// TIA Portal V16 export
// export: Created 2022-11-17T15:49:28.7490525Z, ExportSetting WithDefaults, DisplayName Totally Integrated Automation Portal, DisplayVersion V16 Update 6, DisplayName TIA Portal Version Control Interface, DisplayVersion V16 Update 2, DisplayName TIA Portal Openness, DisplayVersion V16 Update 6, DisplayName SINAMICS Startdrive Advanced, DisplayVersion V16 Update 5, DisplayName SINAMICS Startdrive G130, G150, S120, S150, SINAMICS MV, S210, DisplayVersion V16 Update 5, DisplayName SINAMICS Startdrive G110M, G120, G120C, G120D, G120P, G115D, DisplayVersion V16 Update 5, DisplayName STEP 7 Professional, DisplayVersion V16 Update 6, DisplayName STEP 7 Safety, DisplayVersion V16, DisplayName WinCC Advanced, DisplayVersion V16 Update 6
FUNCTION "FC78_Conveyor_1_IN_1_OUT_REVERSE" : Void   // FC78, LAD
TITLE = Conveyor_1_IN_1_OUT
{ S7_Optimized_Access := 'TRUE' }
VERSION : 0.1
// stored: AutoNumber false, IsIECCheckEnabled false, SetENOAutomatically false, UDAEnableTagReadback false
   VAR_TEMP   // added for the SCL form of the ladder/FBD networks
      _w1 : Bool;
   END_VAR
BEGIN

REGION Network 1: Manual operation for conveyor
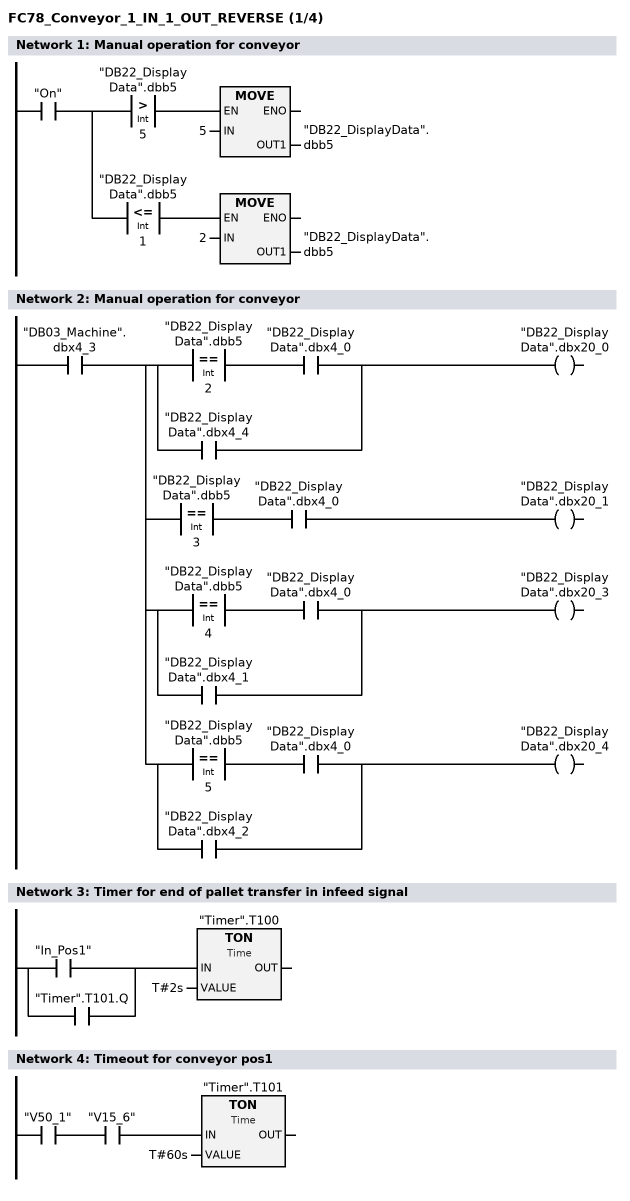
   RUNG wire#powerrail
      Contact( "On" )
      wire#w1
      { S7_Templates := "SrcType := Int" } GT_Contact(in1 := "DB22_DisplayData".dbb5, in2 := 5)
      { S7_GenerateENO := "TRUE" } Move(in := 5, out1 => "DB22_DisplayData".dbb5)
   END_RUNG
   RUNG wire#w1
      { S7_Templates := "SrcType := Int" } LE_Contact(in1 := "DB22_DisplayData".dbb5, in2 := 1)
      { S7_GenerateENO := "TRUE" } Move(in := 2, out1 => "DB22_DisplayData".dbb5)
   END_RUNG
   // the same network as SCL:
   IF "On" AND ("DB22_DisplayData".dbb5 > 5) THEN "DB22_DisplayData".dbb5 := 5; END_IF;
   IF "On" AND ("DB22_DisplayData".dbb5 <= 1) THEN "DB22_DisplayData".dbb5 := 2; END_IF;
END_REGION

REGION Network 2: Manual operation for conveyor
   RUNG wire#powerrail
      Contact( "DB03_Machine".dbx4_3 )
      wire#w1
      { S7_Templates := "SrcType := Int" } EQ_Contact(in1 := "DB22_DisplayData".dbb5, in2 := 2)
      Contact( "DB22_DisplayData".dbx4_0 )
      wire#w2
      Coil( "DB22_DisplayData".dbx20_0 )
   END_RUNG
   RUNG wire#w1
      Contact( "DB22_DisplayData".dbx4_4 )
   END_RUNG wire#w2
   RUNG wire#w1
      { S7_Templates := "SrcType := Int" } EQ_Contact(in1 := "DB22_DisplayData".dbb5, in2 := 3)
      Contact( "DB22_DisplayData".dbx4_0 )
      Coil( "DB22_DisplayData".dbx20_1 )
   END_RUNG
   RUNG wire#w1
      { S7_Templates := "SrcType := Int" } EQ_Contact(in1 := "DB22_DisplayData".dbb5, in2 := 4)
      Contact( "DB22_DisplayData".dbx4_0 )
      wire#w3
      Coil( "DB22_DisplayData".dbx20_3 )
   END_RUNG
   RUNG wire#w1
      Contact( "DB22_DisplayData".dbx4_1 )
   END_RUNG wire#w3
   RUNG wire#w1
      { S7_Templates := "SrcType := Int" } EQ_Contact(in1 := "DB22_DisplayData".dbb5, in2 := 5)
      Contact( "DB22_DisplayData".dbx4_0 )
      wire#w4
      Coil( "DB22_DisplayData".dbx20_4 )
   END_RUNG
   RUNG wire#w1
      Contact( "DB22_DisplayData".dbx4_2 )
   END_RUNG wire#w4
   // the same network as SCL:
   "DB22_DisplayData".dbx20_0 := "DB03_Machine".dbx4_3 AND ((("DB22_DisplayData".dbb5 = 2) AND "DB22_DisplayData".dbx4_0) OR "DB22_DisplayData".dbx4_4);
   "DB22_DisplayData".dbx20_1 := "DB03_Machine".dbx4_3 AND ("DB22_DisplayData".dbb5 = 3) AND "DB22_DisplayData".dbx4_0;
   "DB22_DisplayData".dbx20_3 := "DB03_Machine".dbx4_3 AND ((("DB22_DisplayData".dbb5 = 4) AND "DB22_DisplayData".dbx4_0) OR "DB22_DisplayData".dbx4_1);
   "DB22_DisplayData".dbx20_4 := "DB03_Machine".dbx4_3 AND ((("DB22_DisplayData".dbb5 = 5) AND "DB22_DisplayData".dbx4_0) OR "DB22_DisplayData".dbx4_2);
END_REGION

REGION Network 3: Timer for end of pallet transfer in infeed signal
   "Timer".T100.TON(IN := "In_Pos1" OR "Timer".T101.Q, PT := T#2s);   // TON coil
END_REGION

REGION Network 4: Timeout for conveyor pos1
   "Timer".T101.TON(IN := "V50_1" AND "V15_6", PT := T#60s);   // TON coil
END_REGION

REGION Network 5: Time to load with forklift
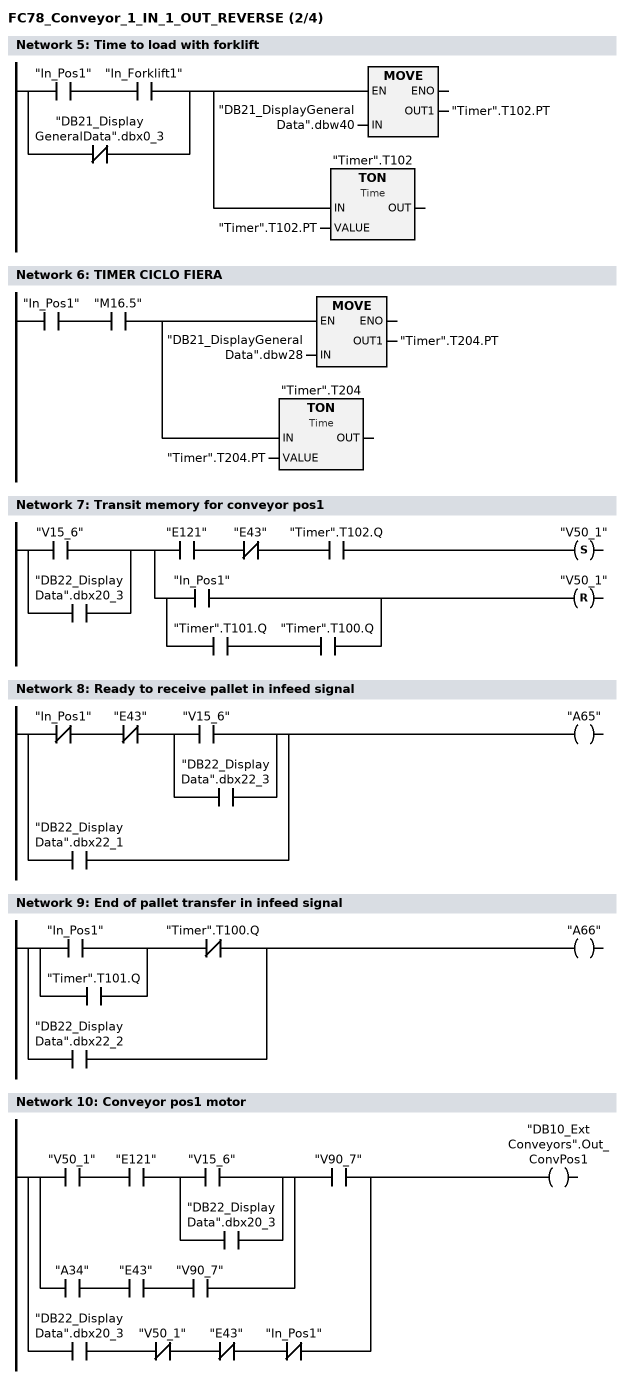
   #_w1 := ("In_Pos1" AND "In_Forklift1") OR NOT "DB21_DisplayGeneralData".dbx0_3;
   IF #_w1 THEN "Timer".T102.PT := "DB21_DisplayGeneralData".dbw40; END_IF;
   "Timer".T102.TON(IN := #_w1, PT := "Timer".T102.PT);   // TON coil
END_REGION

REGION Network 6: TIMER CICLO FIERA
   #_w1 := "In_Pos1" AND "M16.5";
   IF #_w1 THEN "Timer".T204.PT := "DB21_DisplayGeneralData".dbw28; END_IF;
   "Timer".T204.TON(IN := #_w1, PT := "Timer".T204.PT);   // TON coil
END_REGION

REGION Network 7: Transit memory for conveyor pos1
   RUNG wire#powerrail
      Contact( "V15_6" )
      wire#w1
      Contact( "E121" )
      I_Contact( "E43" )
      Contact( "Timer".T102.Q )
      S_Coil( "V50_1" )
   END_RUNG
   RUNG wire#powerrail
      Contact( "DB22_DisplayData".dbx20_3 )
   END_RUNG wire#w1
   RUNG wire#w1
      Contact( "In_Pos1" )
      wire#w2
      R_Coil( "V50_1" )
   END_RUNG
   RUNG wire#w1
      Contact( "Timer".T101.Q )
      Contact( "Timer".T100.Q )
   END_RUNG wire#w2
   // the same network as SCL:
   #_w1 := "V15_6" OR "DB22_DisplayData".dbx20_3;
   IF #_w1 AND "E121" AND NOT "E43" AND "Timer".T102.Q THEN "V50_1" := TRUE; END_IF;
   IF #_w1 AND ("In_Pos1" OR ("Timer".T101.Q AND "Timer".T100.Q)) THEN "V50_1" := FALSE; END_IF;
END_REGION

REGION Network 8: Ready to receive pallet in infeed signal
   RUNG wire#powerrail
      I_Contact( "In_Pos1" )
      I_Contact( "E43" )
      wire#w1
      Contact( "V15_6" )
      wire#w2
      Coil( "A65" )
   END_RUNG
   RUNG wire#w1
      Contact( "DB22_DisplayData".dbx22_3 )
   END_RUNG wire#w2
   RUNG wire#powerrail
      Contact( "DB22_DisplayData".dbx22_1 )
   END_RUNG wire#w2
   // the same network as SCL:
   "A65" := (NOT "In_Pos1" AND NOT "E43" AND ("V15_6" OR "DB22_DisplayData".dbx22_3)) OR "DB22_DisplayData".dbx22_1;
END_REGION

REGION Network 9: End of pallet transfer in infeed signal
   RUNG wire#powerrail
      Contact( "In_Pos1" )
      wire#w1
      I_Contact( "Timer".T100.Q )
      wire#w2
      Coil( "A66" )
   END_RUNG
   RUNG wire#powerrail
      Contact( "Timer".T101.Q )
   END_RUNG wire#w1
   RUNG wire#powerrail
      Contact( "DB22_DisplayData".dbx22_2 )
   END_RUNG wire#w2
   // the same network as SCL:
   "A66" := (("In_Pos1" OR "Timer".T101.Q) AND NOT "Timer".T100.Q) OR "DB22_DisplayData".dbx22_2;
END_REGION

REGION Network 10: Conveyor pos1 motor
   RUNG wire#powerrail
      Contact( "V50_1" )
      Contact( "E121" )
      wire#w1
      Contact( "V15_6" )
      wire#w2
      Contact( "V90_7" )
      wire#w3
      Coil( "DB10_ExtConveyors".Out_ConvPos1 )
   END_RUNG
   RUNG wire#w1
      Contact( "DB22_DisplayData".dbx20_3 )
   END_RUNG wire#w2
   RUNG wire#powerrail
      Contact( "A34" )
      Contact( "E43" )
      Contact( "V90_7" )
   END_RUNG wire#w2
   RUNG wire#powerrail
      Contact( "DB22_DisplayData".dbx20_3 )
      I_Contact( "V50_1" )
      I_Contact( "E43" )
      I_Contact( "In_Pos1" )
   END_RUNG wire#w3
   // the same network as SCL:
   "DB10_ExtConveyors".Out_ConvPos1 := ((("V50_1" AND "E121" AND ("V15_6" OR "DB22_DisplayData".dbx20_3)) OR ("A34" AND "E43" AND "V90_7")) AND "V90_7") OR ("DB22_DisplayData".dbx20_3 AND NOT "V50_1" AND NOT "E43" AND NOT "In_Pos1");
END_REGION

REGION Network 11: Conveyor pos1 motor speed selection
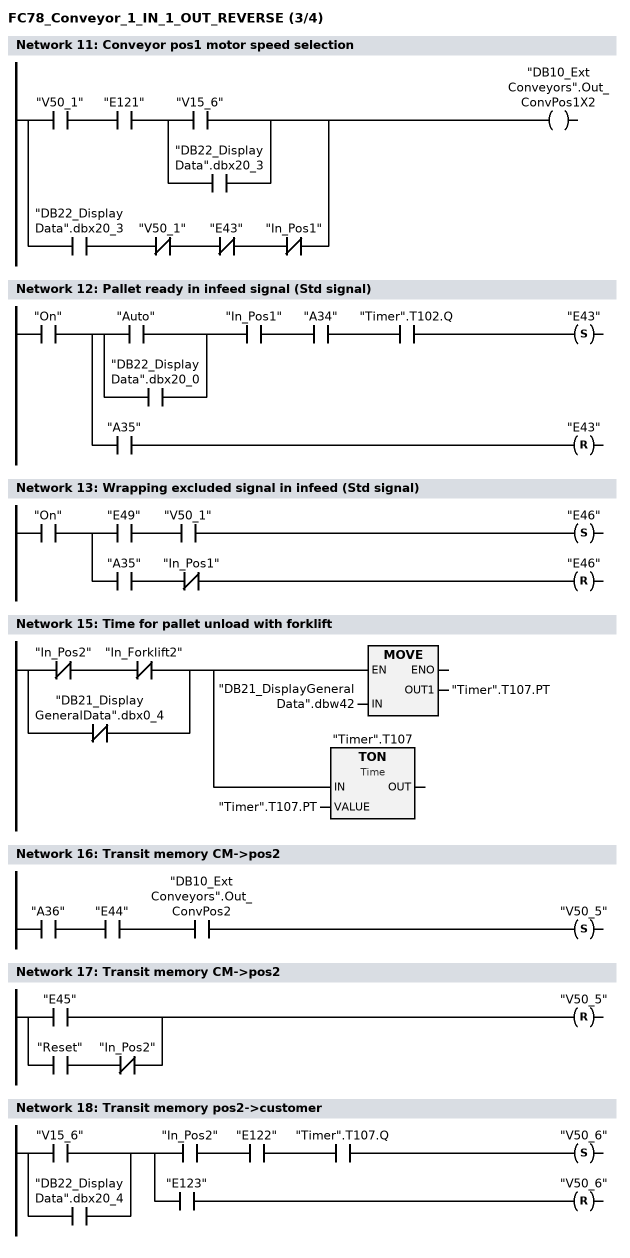
   RUNG wire#powerrail
      Contact( "V50_1" )
      Contact( "E121" )
      wire#w1
      Contact( "V15_6" )
      wire#w2
      Coil( "DB10_ExtConveyors".Out_ConvPos1X2 )
   END_RUNG
   RUNG wire#w1
      Contact( "DB22_DisplayData".dbx20_3 )
   END_RUNG wire#w2
   RUNG wire#powerrail
      Contact( "DB22_DisplayData".dbx20_3 )
      I_Contact( "V50_1" )
      I_Contact( "E43" )
      I_Contact( "In_Pos1" )
   END_RUNG wire#w2
   // the same network as SCL:
   "DB10_ExtConveyors".Out_ConvPos1X2 := ("V50_1" AND "E121" AND ("V15_6" OR "DB22_DisplayData".dbx20_3)) OR ("DB22_DisplayData".dbx20_3 AND NOT "V50_1" AND NOT "E43" AND NOT "In_Pos1");
END_REGION

REGION Network 12: Pallet ready in infeed signal (Std signal)
   RUNG wire#powerrail
      Contact( "On" )
      wire#w1
      Contact( "Auto" )
      wire#w2
      Contact( "In_Pos1" )
      Contact( "A34" )
      Contact( "Timer".T102.Q )
      S_Coil( "E43" )
   END_RUNG
   RUNG wire#w1
      Contact( "DB22_DisplayData".dbx20_0 )
   END_RUNG wire#w2
   RUNG wire#w1
      Contact( "A35" )
      R_Coil( "E43" )
   END_RUNG
   // the same network as SCL:
   IF "On" AND ("Auto" OR "DB22_DisplayData".dbx20_0) AND "In_Pos1" AND "A34" AND "Timer".T102.Q THEN
       "E43" := TRUE;
   END_IF;
   IF "On" AND "A35" THEN "E43" := FALSE; END_IF;
END_REGION

REGION Network 13: Wrapping excluded signal in infeed (Std signal)
   RUNG wire#powerrail
      Contact( "On" )
      wire#w1
      Contact( "E49" )
      Contact( "V50_1" )
      S_Coil( "E46" )
   END_RUNG
   RUNG wire#w1
      Contact( "A35" )
      I_Contact( "In_Pos1" )
      R_Coil( "E46" )
   END_RUNG
   // the same network as SCL:
   IF "On" AND "E49" AND "V50_1" THEN "E46" := TRUE; END_IF;
   IF "On" AND "A35" AND NOT "In_Pos1" THEN "E46" := FALSE; END_IF;
END_REGION

REGION Network 14: >>>>>>> OUTFEED CONVEYOR <<<<<<<<
END_REGION

REGION Network 15: Time for pallet unload with forklift
   #_w1 := (NOT "In_Pos2" AND NOT "In_Forklift2") OR NOT "DB21_DisplayGeneralData".dbx0_4;
   IF #_w1 THEN "Timer".T107.PT := "DB21_DisplayGeneralData".dbw42; END_IF;
   "Timer".T107.TON(IN := #_w1, PT := "Timer".T107.PT);   // TON coil
END_REGION

REGION Network 16: Transit memory CM->pos2
   RUNG wire#powerrail
      Contact( "A36" )
      Contact( "E44" )
      Contact( "DB10_ExtConveyors".Out_ConvPos2 )
      S_Coil( "V50_5" )
   END_RUNG
   // the same network as SCL:
   IF "A36" AND "E44" AND "DB10_ExtConveyors".Out_ConvPos2 THEN "V50_5" := TRUE; END_IF;
END_REGION

REGION Network 17: Transit memory CM->pos2
   RUNG wire#powerrail
      Contact( "E45" )
      wire#w1
      R_Coil( "V50_5" )
   END_RUNG
   RUNG wire#powerrail
      Contact( "Reset" )
      I_Contact( "In_Pos2" )
   END_RUNG wire#w1
   // the same network as SCL:
   IF "E45" OR ("Reset" AND NOT "In_Pos2") THEN "V50_5" := FALSE; END_IF;
END_REGION

REGION Network 18: Transit memory pos2->customer
   RUNG wire#powerrail
      Contact( "V15_6" )
      wire#w1
      Contact( "In_Pos2" )
      Contact( "E122" )
      Contact( "Timer".T107.Q )
      S_Coil( "V50_6" )
   END_RUNG
   RUNG wire#powerrail
      Contact( "DB22_DisplayData".dbx20_4 )
   END_RUNG wire#w1
   RUNG wire#w1
      Contact( "E123" )
      R_Coil( "V50_6" )
   END_RUNG
   // the same network as SCL:
   #_w1 := "V15_6" OR "DB22_DisplayData".dbx20_4;
   IF #_w1 AND "In_Pos2" AND "E122" AND "Timer".T107.Q THEN "V50_6" := TRUE; END_IF;
   IF #_w1 AND "E123" THEN "V50_6" := FALSE; END_IF;
END_REGION

REGION Network 19: Ready to receive pallet from outfeed signal (Signal for Technoplat)
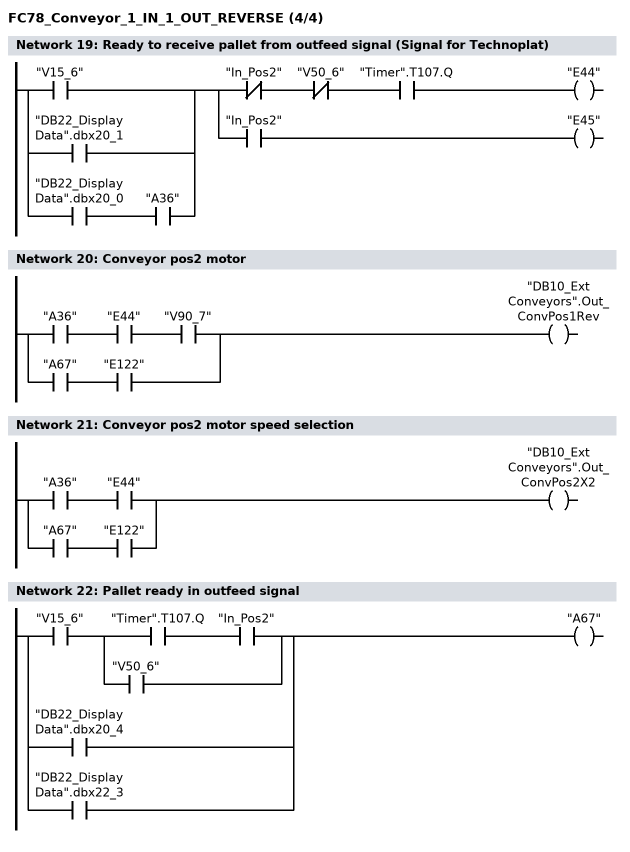
   RUNG wire#powerrail
      Contact( "V15_6" )
      wire#w1
      I_Contact( "In_Pos2" )
      I_Contact( "V50_6" )
      Contact( "Timer".T107.Q )
      Coil( "E44" )
   END_RUNG
   RUNG wire#powerrail
      Contact( "DB22_DisplayData".dbx20_1 )
   END_RUNG wire#w1
   RUNG wire#powerrail
      Contact( "DB22_DisplayData".dbx20_0 )
      Contact( "A36" )
   END_RUNG wire#w1
   RUNG wire#w1
      Contact( "In_Pos2" )
      Coil( "E45" )
   END_RUNG
   // the same network as SCL:
   #_w1 := "V15_6" OR "DB22_DisplayData".dbx20_1 OR ("DB22_DisplayData".dbx20_0 AND "A36");
   "E44" := #_w1 AND NOT "In_Pos2" AND NOT "V50_6" AND "Timer".T107.Q;
   "E45" := #_w1 AND "In_Pos2";
END_REGION

REGION Network 20: Conveyor pos2 motor
   RUNG wire#powerrail
      Contact( "A36" )
      Contact( "E44" )
      Contact( "V90_7" )
      wire#w1
      Coil( "DB10_ExtConveyors".Out_ConvPos1Rev )
   END_RUNG
   RUNG wire#powerrail
      Contact( "A67" )
      Contact( "E122" )
   END_RUNG wire#w1
   // the same network as SCL:
   "DB10_ExtConveyors".Out_ConvPos1Rev := ("A36" AND "E44" AND "V90_7") OR ("A67" AND "E122");
END_REGION

REGION Network 21: Conveyor pos2 motor speed selection
   RUNG wire#powerrail
      Contact( "A36" )
      Contact( "E44" )
      wire#w1
      Coil( "DB10_ExtConveyors".Out_ConvPos2X2 )
   END_RUNG
   RUNG wire#powerrail
      Contact( "A67" )
      Contact( "E122" )
   END_RUNG wire#w1
   // the same network as SCL:
   "DB10_ExtConveyors".Out_ConvPos2X2 := ("A36" AND "E44") OR ("A67" AND "E122");
END_REGION

REGION Network 22: Pallet ready in outfeed signal
   RUNG wire#powerrail
      Contact( "V15_6" )
      wire#w1
      Contact( "Timer".T107.Q )
      Contact( "In_Pos2" )
      wire#w2
      Coil( "A67" )
   END_RUNG
   RUNG wire#w1
      Contact( "V50_6" )
   END_RUNG wire#w2
   RUNG wire#powerrail
      Contact( "DB22_DisplayData".dbx20_4 )
   END_RUNG wire#w2
   RUNG wire#powerrail
      Contact( "DB22_DisplayData".dbx22_3 )
   END_RUNG wire#w2
   // the same network as SCL:
   "A67" := ("V15_6" AND (("Timer".T107.Q AND "In_Pos2") OR "V50_6")) OR "DB22_DisplayData".dbx20_4 OR "DB22_DisplayData".dbx22_3;
END_REGION
END_FUNCTION
